PROGRAM MAIN
VAR
END_VAR

prgAlarms();

END_PROGRAM

(* stored: Version 1.1.0.1, ProductVersion 3.1.4024.11
   POU MAIN: Id {5d50a675-cd2a-48b8-81e1-295a6a0df70b}, SpecialFunc None *)
